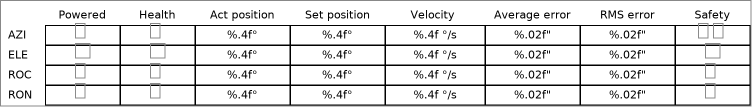
VISUALIZATION VISU_Axes_stats  // 752x107
VAR_IN_OUT
	ref : Axes;
    widget : AxesWidget;
END_VAR
    Rectangle (675,85 75x20)
    Rectangle (675,45 75x20)
    Rectangle (675,65 75x20)
    Rectangle (675,25 75x20)
    Rectangle (45,85 75x20)
    Rectangle (45,45 75x20)
    Rectangle (45,65 75x20)
    Rectangle (45,25 75x20)
    Rectangle (485,25 95x20), "%.02f"", text variable: ref.parts.azi.deviation1SecAverage.arcseconds.value
    Label (485,5 95x20), "Average error"
    Rectangle (580,25 95x20), "%.02f"", text variable: ref.parts.azi.deviation1SecRMS.arcseconds.value
    Rectangle (485,45 95x20), "%.02f"", text variable: ref.parts.ele.deviation1SecAverage.arcseconds.value
    Label (5,25 40x20), "AZI"
    Label (5,45 40x20), "ELE"
    Rectangle (580,45 95x20), "%.02f"", text variable: ref.parts.ele.deviation1SecRMS.arcseconds.value
    Label (580,5 95x20), "RMS error"
    Rectangle (485,65 95x20), "%.02f"", text variable: ref.parts.roc.deviation1SecAverage.arcseconds.value
    Rectangle (580,65 95x20), "%.02f"", text variable: ref.parts.roc.deviation1SecRMS.arcseconds.value
    Rectangle (485,85 95x20), "%.02f"", text variable: ref.parts.ron.deviation1SecAverage.arcseconds.value
    Rectangle (580,85 95x20), "%.02f"", text variable: ref.parts.ron.deviation1SecRMS.arcseconds.value
    Label (5,65 40x20), "ROC"
    Label (5,85 40x20), "RON"
    Label (45,5 75x20), "Powered"
    Frame (75,23 10x15)
        shows VISU_State_gray_green(state := ref.parts.azi.statuses.poweredStatus.enabled)
    Frame (75,43 15x15)
        shows VISU_State_gray_green(state := ref.parts.ele.statuses.poweredStatus.enabled)
    Frame (75,63 10x15)
        shows VISU_State_gray_green(state := ref.parts.roc.statuses.poweredStatus.enabled)
    Frame (75,83 10x15)
        shows VISU_State_gray_green(state := ref.parts.ron.statuses.poweredStatus.enabled)
    Rectangle (195,25 95x20), "%.4f°", text variable: ref.parts.azi.actPos.degrees.value
    Label (195,5 95x20), "Act position"
    Rectangle (195,45 95x20), "%.4f°", text variable: ref.parts.ele.actPos.degrees.value
    Rectangle (195,65 95x20), "%.4f°", text variable: ref.parts.roc.actPos.degrees.value
    Rectangle (195,85 95x20), "%.4f°", text variable: ref.parts.ron.actPos.degrees.value
    Rectangle (385,25 100x20), "%.4f °/s", text variable: ref.parts.azi.actVelo.degreesPerSecond.value
    Label (385,5 95x20), "Velocity"
    Rectangle (385,45 100x20), "%.4f °/s", text variable: ref.parts.ele.actVelo.degreesPerSecond.value
    Rectangle (385,65 100x20), "%.4f °/s", text variable: ref.parts.roc.actVelo.degreesPerSecond.value
    Rectangle (385,85 100x20), "%.4f °/s", text variable: ref.parts.ron.actVelo.degreesPerSecond.value
    Label (675,5 75x20), "Safety"
    Frame (698,23 10x15)
        shows VISU_State_green_red(state := ref.parts.io.parts.aziDrive.parts.channelA.isInSafetate)
    Frame (705,43 15x15)
        shows VISU_State_green_red(state := ref.parts.io.parts.eleDrive.parts.channelA.isInSafetate)
    Frame (705,63 10x15)
        shows VISU_State_green_red(state := ref.parts.io.parts.aziDrive.parts.channelB.isInSafetate)
    Frame (705,83 10x15)
        shows VISU_State_green_red(state := ref.parts.io.parts.ablDrive.parts.channelB.isInSafetate)
    Frame (713,23 10x15)
        shows VISU_State_green_red(state := ref.parts.io.parts.ablDrive.parts.channelA.isInSafetate)
    Rectangle (290,25 95x20), "%.4f°", text variable: ref.parts.azi.setPos.degrees.value
    Label (290,5 95x20), "Set position"
    Rectangle (290,45 95x20), "%.4f°", text variable: ref.parts.ele.setPos.degrees.value
    Rectangle (290,65 95x20), "%.4f°", text variable: ref.parts.roc.setPos.degrees.value
    Rectangle (290,85 95x20), "%.4f°", text variable: ref.parts.ron.setPos.degrees.value
    Rectangle (120,85 75x20)
    Rectangle (120,45 75x20)
    Rectangle (120,65 75x20)
    Rectangle (120,25 75x20)
    Label (120,5 75x20), "Health"
    Frame (150,43 15x15)
        shows VISU_State_green_red(state := ref.parts.ele.statuses.healthStatus.bad)
    Frame (150,63 10x15)
        shows VISU_State_green_red(state := ref.parts.roc.statuses.healthStatus.bad)
    Frame (150,83 10x15)
        shows VISU_State_green_red(state := ref.parts.ron.statuses.healthStatus.bad)
    Frame (150,23 10x15)
        shows VISU_State_green_red(state := ref.parts.azi.statuses.healthStatus.bad)
END_VISUALIZATION

(* stored: Version 1.1.0.1, ProductVersion 3.1.4019.2
   Visu VISU_Axes_stats: Id {2768193e-041c-44ae-8e9b-71ed5b6e0964} *)
